TYPE E_FunctionType :
(
	eSine,
	eSquare,
	ePulse,
	eTriangular,
	eSawtooth,	
	eAM
);
END_TYPE

(* stored: Version 1.1.0.1, ProductVersion 3.1.4022.12
   DUT E_FunctionType: Id {417c2037-ff55-4eac-9eb2-4a287a02424d} *)
